FUNCTION_BLOCK SET_LTIME (* Writes a LTIME value from an Input to an InOut variable *)
  (* Standard: 61499-1 *)
  (* Version 1.0, 2026-05-07, Gemini CLI, Initial version *)
  PACKAGE logiBUS::utils::conversion::provide;
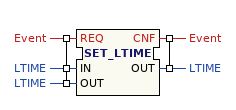
  EVENT_INPUT
    REQ WITH IN, OUT; (* Normal Execution Request *)
  END_EVENT
  EVENT_OUTPUT
    CNF WITH OUT; (* Execution Confirmation *)
  END_EVENT
  VAR_INPUT
    IN : LTIME := LT#0s; (* Value to be written *)
  END_VAR
  VAR_IN_OUT
    OUT : LTIME := LT#0s; (* Target variable (InOut) *)
  END_VAR
  EC_STATES
    REQ : REQ -> CNF;
  END_STATES
  ALGORITHM REQ IN ST: (* Write input value to the InOut target variable *)
OUT := IN;
  END_ALGORITHM
END_FUNCTION_BLOCK
